INTERFACE I_STREAM

PROPERTY BufferSize : UDINT
GET
END_GET
END_PROPERTY

METHOD Close : DINT
VAR_INPUT
END_VAR
END_METHOD

PROPERTY EndOfStream : BOOL
GET
END_GET
END_PROPERTY

PROPERTY IsValid : BOOL
GET
END_GET
END_PROPERTY

METHOD Peek : DINT
VAR_INPUT
	ptr_DataOut : POINTER TO BYTE;
END_VAR
END_METHOD

PROPERTY Position : UDINT
GET
END_GET
END_PROPERTY

METHOD Read : DINT
VAR_INPUT
	ptr_DataOut : PVOID;
	Length		: UDINT;
END_VAR
END_METHOD

METHOD Seek : DINT
VAR_INPUT
	Offset 		: UDINT;
	SeekStyle 	: E_STREAMSEEKTYPE;
END_VAR
END_METHOD

METHOD Write : DINT
VAR_INPUT
	ptr_DataIn	: PVOID;
	Length		: UDINT;
END_VAR
END_METHOD

END_INTERFACE

(* stored: Version 1.1.0.1, ProductVersion 3.1.4022.3
   Itf I_STREAM: Id {de9b42df-215f-45d1-a5c2-a220dc4efd75}
   Folder Methods: Id {56321ced-c9b4-4c73-9f76-c8870b997027}
   Folder Properties: Id {fcc502e0-de76-4dda-8f16-1ee84b9c58df}
   Property BufferSize: Id {8d9ad315-d518-4be2-9664-ecb88a70d6d9}
   Get Get: Id {2271780a-fd91-4755-bd0d-ca0a3ef46b5b}
   Method Close: Id {a0f98e8a-e3e3-450e-bb2f-9220cb3d18ea}
   Property EndOfStream: Id {accf14f5-c45c-4747-b268-b60455de1537}
   Get Get: Id {d7f24878-c874-4c7a-bf53-23151ae3ef62}
   Property IsValid: Id {f5a40038-c188-4112-afb9-225d644d66b4}
   Get Get: Id {5d9a6a82-1282-40a9-833f-c0ec844eac26}
   Method Peek: Id {e44c98bf-5c46-48fd-a256-068e26b8a34e}
   Property Position: Id {52cb7e0a-7f61-4e73-9715-280da83f2fbe}
   Get Get: Id {baf57325-0a65-4495-af0b-eb19d902b6f6}
   Method Read: Id {f2133b03-4975-487a-a57f-516773cc13e2}
   Method Seek: Id {411ab45e-ced1-4733-b80d-19981489e95a}
   Method Write: Id {a10e8fa8-d36b-4ede-8694-1b43b82478c3} *)
